PROGRAM MAIN
VAR
END_VAR

END_PROGRAM

(* stored: Version 1.1.0.1
   POU MAIN: Id {e4e8c683-e553-4ffa-9f26-b8cf7ac5125a} *)
